ABB RobotStudio station: Socket_Communication.rspag

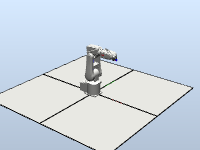
--- station ---
Station Socket_Communication (saved by RobotStudio 6.8.8148.134)
Controller IRB_120_3kg_0.58m
  mechanical unit ROB_1: IRB120_3_58__01, 6 joints, base frame (0, 0, 0) mm
Layout (positions relative to the parent item):
  - IRB120_3_58__01 [mechanism, from Robots\IRB120_3_58_G_01.rslib] at (0, 0, 0) mm; joint values [0, 0, 0, 0, 0.5236, 0] (rad or m)

--- Backups/IRB_120_3kg_0.58m/RAPID/TASK1/PROGMOD/Module1.mod ---
MODULE Module1
    VAR socketdev serverSocket;
    VAR socketdev clientSocket;
    VAR string data;

    PROC main()
        SocketCreate serverSocket;
        SocketBind serverSocket,"127.0.0.1",4000;
        SocketListen serverSocket;
        SocketAccept serverSocket,clientSocket,\Time:=WAIT_MAX;

        WHILE TRUE DO

            SocketReceive clientSocket\Str:=data;       ! from C# app
            SocketSend clientSocket\Str:=data + "_";    ! to C# app

        ENDWHILE

        SocketClose clientSocket;
        SocketClose serverSocket;

    ERROR

        IF ERRNO=ERR_SOCK_TIMEOUT THEN
            RETRY;

        ELSEIF ERRNO=ERR_SOCK_CLOSED THEN
            SocketClose clientSocket;

            SocketClose serverSocket;
            SocketCreate serverSocket;
            SocketBind serverSocket,"127.0.0.1",4000;
            SocketListen serverSocket;
            SocketAccept serverSocket,clientSocket,\Time:=WAIT_MAX;

            RETRY;

        ELSE
            stop;
        ENDIF

    ENDPROC
ENDMODULE
